FUNCTION_BLOCK FB_StateMachine1 EXTENDS FB_StateMachine
VAR_INPUT
END_VAR
VAR_OUTPUT
END_VAR
VAR
END_VAR

END_FUNCTION_BLOCK

(* stored: Version 1.1.0.1, ProductVersion 3.1.4024.12
   POU FB_StateMachine1: Id {42eb1aad-753e-44e4-851c-8bc02a4713ae}, SpecialFunc None *)
